TYPE ST_HMI_PACK_BufferStatus :
STRUCT
	nPacksPerOuter				: INT;
	nMaxPackPerOuter				: INT;
	aPackBuffer1					: ARRAY[1..cMAX_HMI_PACKS_PER_OUTER] OF ST_HMI_OCV_Data;
	aPackBuffer2					: ARRAY[1..cMAX_HMI_PACKS_PER_OUTER] OF ST_HMI_OCV_Data;
END_STRUCT
END_TYPE

(* stored: Version 1.1.0.1
   DUT ST_HMI_PACK_BufferStatus: Id {084c2d12-a0bf-4a4b-ac98-dbaf650ed079} *)
